(* IEC 61131-3 sources: string-builder/src, 4 files *)

(* ---- IConstrainedStringBuilder.st ---- *)
NAMESPACE Simatic.Ax.Strings
    INTERFACE IConstrainedStringBuilder
        METHOD Append : IStringBuilder
            VAR_INPUT
                t : STRING;
            END_VAR
        END_METHOD

        METHOD Reset : IConstrainedStringBuilder END_METHOD

        METHOD ToString : STRING END_METHOD
    END_INTERFACE
END_NAMESPACE

(* ---- IStringBuilder.st ---- *)
NAMESPACE Simatic.Ax.Strings
    INTERFACE IStringBuilder EXTENDS IConstrainedStringBuilder
        METHOD Insert : IStringBuilder
            VAR_INPUT
                t : STRING;
                pos : INT;
            END_VAR
        END_METHOD

        METHOD Remove : IStringBuilder
            VAR_INPUT
                t: STRING;
                startPos : INT;
                length : INT;
            END_VAR
        END_METHOD

        METHOD Substring : IStringBuilder
            VAR_INPUT
                t : STRING;
                startPos : INT;
                length : INT;
            END_VAR
        END_METHOD

        METHOD  StartOf : IStringBuilder
            VAR_INPUT
                t : STRING;
                length : INT;
            END_VAR
        END_METHOD

        METHOD  EndOf : IStringBuilder
            VAR_INPUT
                t : STRING;
                length : INT;
            END_VAR
        END_METHOD

        METHOD Replace : IStringBuilder
            VAR_INPUT
                t : STRING;
                startPos : INT;
                length : INT;
                replaceValue : STRING;
            END_VAR
        END_METHOD
    END_INTERFACE
END_NAMESPACE

(* ---- myClass.st ---- *)
NAMESPACE Simatic.Ax.string-builder

    {axcode:docs-v0:@simatic-ax/string-builder:MyClass.md}
    CLASS MyClass

        VAR PUBLIC
        END_VAR

        VAR
        END_VAR

        /// Inline Comment for MyMethod. It will be shown, when you hover over the method
        /// This method has no parameters and no return value
        METHOD PUBLIC MyMethod
            ;
        END_METHOD

    END_CLASS

END_NAMESPACE

(* ---- StringBuilder.st ---- *)
USING System.Strings;
NAMESPACE Simatic.Ax.Strings
    CLASS StringBuilder IMPLEMENTS IStringBuilder, IConstrainedStringBuilder
        VAR
            _string : STRING;
        END_VAR

        METHOD PUBLIC Append : IStringBuilder
            VAR_INPUT
                t : STRING;
            END_VAR
            _string := Concat(_string, t);
            Append := THIS;
        END_METHOD

        METHOD PUBLIC Insert : IStringBuilder
            VAR_INPUT
                t : STRING;
                pos : INT;
            END_VAR
            _string := Insert(_string, pos, t);
            Insert := THIS;
        END_METHOD

        METHOD PUBLIC Reset : IConstrainedStringBuilder
            _string := '';
            Reset := THIS;
        END_METHOD

        METHOD PUBLIC ToString : STRING
            ToString := _string;
        END_METHOD

        METHOD PUBLIC Remove : IStringBuilder
            VAR_INPUT
                t : STRING;
                startPos : INT;
                length : INT;
            END_VAR
            _string := Remove(t, startPos, length);
            Remove := THIS;
        END_METHOD

        METHOD PUBLIC Substring : IStringBuilder
            VAR_INPUT
                t : STRING;
                startPos : INT;
                length : INT;
            END_VAR
            _string := Substring(t, startPos, length);
            Substring := THIS;
        END_METHOD

        METHOD PUBLIC StartOf : IStringBuilder
            VAR_INPUT
                t : STRING;
                length : INT;
            END_VAR
            _string := StartOf(t, length);
            StartOf := THIS;
        END_METHOD

        METHOD PUBLIC Replace : IStringBuilder
            VAR_INPUT
                t : STRING;
                startPos : INT;
                length : INT;
                replaceValue : STRING;
            END_VAR
            _string := Replace(t, startPos, length, replaceValue);
            Replace := THIS;
        END_METHOD

        METHOD PUBLIC EndOf : IStringBuilder
            VAR_INPUT
                t : STRING;
                length : INT;
            END_VAR
            _string := EndOf(t, length);
            EndOf := THIS;
        END_METHOD
    END_CLASS
END_NAMESPACE
